PROPERTY IsClosed : BOOL
GET
IF ipTrack <> 0 THEN
	IsClosed := ipTrack.GetIsClosed();
ELSE
	Trace('IsClosed called before initialization!');
	_Error := TRUE;
END_IF
END_GET
END_PROPERTY

PROPERTY Length : LREAL
GET
IF ipTrack <> 0 THEN
	Length := ipTrack.GetLength();
ELSE
	Trace('Length called before initialization!');
	_Error := TRUE;
END_IF
END_GET
END_PROPERTY

PROPERTY Name : STRING
GET
IF ipTrack <> 0 THEN
	Name := ipTrack.GetObjectName();
ELSE
	Trace('Name called before initialization!');
	_Error := TRUE;
END_IF
END_GET
END_PROPERTY

METHOD PRIVATE Initialize : BOOL
CASE InitializeState OF
	E_InitializeState_Track.eInitializeStateTrack_Check:
		IF ipTrack <> 0 THEN
			InitializeState := E_InitializeState_Track.eInitializeStateTrack_GetPartInfo;
		ELSE
			IF Parameters_XTS.ENABLE_DEBUG_TRACING THEN
				Trace('Track initialization attempted with null reference');
			END_IF

			InitializeState := E_InitializeState_Track.eInitializeStateTrack_Failed;
		END_IF

	E_InitializeState_Track.eInitializeStateTrack_GetPartInfo:
		NumberOfParts := ipTrack.GetPartCount();
		Parts		  REF= ipTrack.GetPartInfoItems();
		IF NumberOfParts = 0 THEN
			IF Parameters_XTS.ENABLE_DEBUG_TRACING THEN
				Trace('No parts associated with this track');
			END_IF

			InitializeState := E_InitializeState_Track.eInitializeStateTrack_Failed;
		ELSE
			InitializeState := E_InitializeState_Track.eInitializeStateTrack_Complete;
		END_IF

	E_InitializeState_Track.eInitializeStateTrack_Complete:
		_Busy	   := FALSE;
		Initialize := TRUE;

	E_InitializeState_Track.eInitializeStateTrack_Failed:
		_Busy  := FALSE;
		_Error := TRUE;
END_CASE
END_METHOD

END_FUNCTION_BLOCK

// Utilities/FB_TrackingRegister_Stations
FUNCTION_BLOCK FB_TrackingRegister_Stations
VAR
	Status			 : ARRAY[1..TcIoXtsEnvironmentParameterList.MaxXtsInfoStation] OF BOOL;
	_StationsToTrack : REFERENCE TO UDINT;
END_VAR

//This FB is just for ease of tracking what group commands

//have actually completed

METHOD Check : BOOL
VAR_INPUT
	i : UDINT;
END_VAR
IF __ISVALIDREF(_StationsToTrack) THEN
	IF (i >= 1) AND (i <= _StationsToTrack) THEN
		Check := Status[i];
	END_IF
END_IF
END_METHOD

METHOD Clear : BOOL
MEMSET(ADR(Status), 0, SIZEOF(Status));
END_METHOD

PROPERTY Complete : BOOL
GET
VAR
	i : UDINT;
END_VAR

//Returns true if all operations have completed
IF __ISVALIDREF(_StationsToTrack) THEN
	FOR i := 1 TO _StationsToTrack DO
		IF NOT Status[i] THEN
			Complete := FALSE;
			RETURN;
		END_IF
	END_FOR

	Complete := TRUE;
END_IF
END_GET
END_PROPERTY

PROPERTY NumberCompleted : UDINT
GET
VAR
	i : UDINT;
END_VAR
IF __ISVALIDREF(_StationsToTrack) THEN
	FOR i := 1 TO _StationsToTrack DO
		IF Status[i] THEN
			NumberCompleted := NumberCompleted + 1;
		END_IF
	END_FOR
END_IF
END_GET
END_PROPERTY

METHOD Reset : BOOL
VAR_INPUT
	i : UDINT;
END_VAR
IF __ISVALIDREF(_StationsToTrack) THEN
	IF (i >= 1) AND (i <= _StationsToTrack) THEN
		Status[i] := FALSE;
	END_IF
END_IF
END_METHOD

METHOD Set : BOOL
VAR_INPUT
	i : UDINT;
END_VAR
IF __ISVALIDREF(_StationsToTrack) THEN
	IF (i >= 1) AND (i <= _StationsToTrack) THEN
		Status[i] := TRUE;
	END_IF
END_IF
END_METHOD

PROPERTY StationsToTrack : REFERENCE TO UDINT
GET
StationsToTrack REF= _StationsToTrack;
END_GET
SET
_StationsToTrack REF= StationsToTrack;
END_SET
END_PROPERTY

END_FUNCTION_BLOCK

// XPU/FB_Component_XPU
FUNCTION_BLOCK FINAL FB_Component_XPU EXTENDS FB_ComponentBase IMPLEMENTS I_XTS_Xpu
VAR
	XPUAlarms						: ARRAY[1..CONSTANTS.XPU_ALARM_COUNT] OF FB_TcAlarm;
	CAGroup							: AXES_GROUP_REF; //***Must be linked to the CA group in NC***
	ipXPU							: I_TcIoXtsProcessingUnit;
	ipMc2CAGroup					: I_Mc2CaGroup;
	NumberOfParts					: UDINT;
	Parts							: ARRAY[0..TcIoXtsEnvironmentParameterList.MaxXtsPartsPerXpu] OF FB_XTS_Part;
	NumberOfTracks					: UDINT;
	Tracks							: ARRAY[0..TcIoXtsEnvironmentParameterList.MaxXtsTracksPerXpu] OF FB_XTS_Track;
	NumberOfMovers					: UDINT;
	Movers							: ARRAY[0..TcIoXtsEnvironmentParameterList.MaxXtsMoversPerXpu] OF FB_XTS_Mover;
	ipMovers						: ARRAY[0..TcIoXtsEnvironmentParameterList.MaxXtsMoversPerXpu] OF I_XTS_Mover;
	NumberOfStations				: UDINT;
	InfoStations					: ARRAY[0..TcIoXtsEnvironmentParameterList.MaxXtsInfoServer * TcIoXtsEnvironmentParameterList.MaxXtsInfoStation] OF FB_XTS_InfoStation;
	ipStations						: ARRAY[0..TcIoXtsEnvironmentParameterList.MaxXtsInfoServer * TcIoXtsEnvironmentParameterList.MaxXtsInfoStation] OF I_XTS_ApplicationStation;
	SequenceState					: UDINT;
	InitializeState					: E_XPUInitializeState;
	InitializeState_Environment		: E_XPUInitializeState_Environment;
	InitializeState_XPU				: E_XPUInitializeState_XPU;
	InitializeState_CAGroups		: E_XPUInitializeState_CAGroups;
	InitializeState_InfoStations	: E_XPUInitializeState_InfoStations;
	_State							: E_XTSState;
	MCGroupEnable					: MC_GroupEnable;
	MCGroupDisable					: MC_GroupDisable;
	MCGroupReset					: MC_GroupReset;
	MCGroupStop						: MC_GroupStop;
	MCGroupReadError				: MC_GroupReadError;
	MCGroupReadStatus				: MC_GroupReadStatus;
	MCUngroupAllAxes				: MC_UngroupAllAxes;
	JsonParser						: FB_JsonDomParser;
	MoverTracker					: FB_TrackingRegister_Movers;
	StationTracker					: FB_TrackingRegister_Stations;
	StationRecoveryComplete			: BOOL;
	_MoverAssignmentStorageLocation : E_MoverAssignmentRecoverySource := E_MoverAssignmentRecoverySource.eMoverAssignmentRecoverySource_NoBackup;
	WritePersistentData				: FB_WritePersistentData;
	_PartCoEData					: ARRAY[1..TcIoXtsEnvironmentParameterList.MaxXtsPartsPerXpu] OF ARRAY[1..TcIoXtsEnvironmentParameterList.MaxModulesPerPart] OF ST_AT2xxxAllCoEData;
END_VAR

VAR
	//Upstream/Downstream relationships between stations
	StationNeigbors : ARRAY[0..TcIoXtsEnvironmentParameterList.MaxXtsInfoServer * TcIoXtsEnvironmentParameterList.MaxXtsInfoStation] OF ST_StationNeighbors;
END_VAR

VAR PERSISTENT
	//Power-up mover-station assignments (_MoverAssignmentStorageLocation = E_MoverAssignmentRecoverySource.eMoverAssignmentRecoverySource_Persistent)
	MoverAssignments_Persistent : ARRAY[1..TcIoXtsEnvironmentParameterList.MaxXtsInfoServer * TcIoXtsEnvironmentParameterList.MaxXtsInfoStation] OF ST_MoverAssignmentData;
END_VAR

VAR RETAIN
	//Power-up mover-station assignments (_MoverAssignmentStorageLocation = E_MoverAssignmentRecoverySource.eMoverAssignmentRecoverySource_NOVRAM)
	MoverAssignments_NOVRAM : ARRAY[1..TcIoXtsEnvironmentParameterList.MaxXtsInfoServer * TcIoXtsEnvironmentParameterList.MaxXtsInfoStation] OF ST_MoverAssignmentData;
END_VAR

//! @summary This method serves as the entry point for all underlying FB logic
METHOD PUBLIC CyclicLogic
//! @description This method should be called cyclically by descendant function blocks by invoking <c>SUPER^.CyclicLogic()</c>.  Alternatively, the contents of this method could be reimplemented entirely in which case a call to this method would not be necessary.
VAR
	i, j : UDINT;
END_VAR
SUPER^.CyclicLogic();
IF NOT _InitComplete THEN
	RETURN;
END_IF

FOR i := 1 TO NumberOfParts DO
	Parts[i].CyclicLogic();
	IF NOT InSimulationMode THEN
		_PartCoEData[i] := Parts[i].ModuleCoEData;
	END_IF
END_FOR

FOR i := 1 TO NumberOfTracks DO
	Tracks[i].CyclicLogic();
END_FOR

FOR i := 1 TO NumberOfMovers DO
	IF ipMovers[i] <> 0 THEN
		ipMovers[i].CyclicLogic();
	END_IF

	FOR j := 1 TO NumberOfParts DO
		IF Movers[i].CurrentPartOID = Parts[j].OID THEN
			Movers[i].CurrentPart := Parts[j];
			EXIT;
		END_IF
	END_FOR

	FOR j := 1 TO NumberOfTracks DO
		IF Movers[i].CurrentTrackOID = Tracks[j].OID THEN
			Movers[i].CurrentTrack := Tracks[j];
			EXIT;
		END_IF
	END_FOR
END_FOR

FOR i := 1 TO NumberOfStations DO
	InfoStations[i].CyclicLogic();
END_FOR

IF StationRecoveryComplete THEN
	CollectRecoveryData();
END_IF

(****************    Call misc. group FBs    ****************)
MCGroupEnable(AxesGroup := CAGroup);
MCGroupDisable(AxesGroup := CAGroup);
MCGroupReset(AxesGroup := CAGroup);
MCGroupStop(AxesGroup := CAGroup);
MCUngroupAllAxes(AxesGroup := CAGroup);
MCGroupReadStatus(AxesGroup := CAGroup, Enable := TRUE);
MCGroupReadError(AxesGroup := CAGroup, Enable := TRUE);
_Busy := (_State <> E_XTSState.eXTSState_Disabled) AND (_State <> E_XTSState.eXTSState_Error) AND (_State <> E_XTSState.eXTSState_Enabled);
END_METHOD

METHOD GetPositionOnTrack : LREAL
VAR_INPUT
	TrackID	 : OTCID;
	PartID	 : OTCID;
	Position : LREAL;
END_VAR

VAR
	i			   : UDINT;
	PositionResult : LREAL;
END_VAR
IF TrackID <> 0 THEN
	FOR i := 1 TO NumberOfTracks DO
		IF Tracks[i].OID = TrackID THEN
			Tracks[i].GetTrackPositionByPart(Position, PartID, TrackPosition => GetPositionOnTrack);
			EXIT;
		END_IF
	END_FOR
ELSE
	Tracks[1].GetTrackPositionByPart(Position, PartID, TrackPosition => GetPositionOnTrack);
END_IF
END_METHOD

METHOD GiveMover : BOOL
VAR_INPUT
	RequestingStation : I_XTS_StationNeighbor;
END_VAR

VAR
	i : UDINT;
END_VAR
FOR i := 0 TO NumberOfStations DO
	IF StationNeigbors[i].Station <> 0 THEN
		IF StationNeigbors[i].Station = RequestingStation THEN
			GiveMover := StationNeigbors[i].UpstreamStation.GiveMover(RequestingStation);
			EXIT;
		END_IF
	END_IF
END_FOR
END_METHOD

PROPERTY InSimulationMode : BOOL
GET
IF ipXPU <> 0 THEN
	InSimulationMode := ipXPU.GetOperationMode() = OperationMode.Simulation;
END_IF
END_GET
END_PROPERTY

//! @summary Initializes event function blocks using this components's name
{attribute 'call_after_online_change_slot' := '<slot>'}
METHOD PROTECTED CreateEvents
VAR
	Temp : STRING;
END_VAR
Temp := CONCAT(CONCAT(CONCAT('XPU', ': '), Name),
			   ' '); //Creates a utility string for alarms and other messaging that reads (example text) - "Module 10 - Main Casepacker" to be followed by the alarm or message info

F_CreateAllEventsInClass(Alarms		:= XPUAlarms,
						 ClassSize	:= SIZEOF(TC_EVENTS.XPUAlarms),
						 pInitEvent := ADR(TC_EVENTS.XPUAlarms.InitReferenceEvent),
						 Prefix		:= Name);

SUPER^.CreateEvents();
END_METHOD

//! Provides basic error detection and event handling for this component
METHOD PROTECTED Monitoring
VAR
	i			  : UDINT;
	FaultsCleared : BOOL;
END_VAR
SUPER^.Monitoring();

//ErrorID 2 - Part Error
FaultsCleared := TRUE;
FOR i := 1 TO NumberOfParts DO
	IF Parts[i].Error THEN
		IF NOT XPUAlarms[E_XPUAlarms.PartError].bRaised THEN
			RaiseAlarmWithStrings(XPUAlarms[E_XPUAlarms.PartError], TO_STRING(i), TO_STRING(Parts[i].ErrorID));
			SetError(Parts[i].ErrorID);
			_State := E_XTSState.eXTSState_Error;
		END_IF

		FaultsCleared := FALSE;
		EXIT;
	END_IF
END_FOR

IF XPUAlarms[E_XPUAlarms.PartError].bRaised AND FaultsCleared THEN
	XPUAlarms[E_XPUAlarms.PartError].Clear(0, 0);
END_IF

//ErrorID 3 - Track Error
FaultsCleared := TRUE;
FOR i := 1 TO NumberOfTracks DO
	IF Tracks[i].Error THEN
		IF NOT XPUAlarms[E_XPUAlarms.TrackError].bRaised THEN
			RaiseAlarmWithStrings(XPUAlarms[E_XPUAlarms.TrackError], TO_STRING(i), TO_STRING(Tracks[i].ErrorID));
			SetError(Tracks[i].ErrorID);
			_State := E_XTSState.eXTSState_Error;
		END_IF

		FaultsCleared := FALSE;
		EXIT;
	END_IF
END_FOR

IF XPUAlarms[E_XPUAlarms.TrackError].bRaised AND FaultsCleared THEN
	XPUAlarms[E_XPUAlarms.TrackError].Clear(0, 0);
END_IF

//ErrorID 4 - Mover Error
FaultsCleared := TRUE;
FOR i := 1 TO NumberOfMovers DO
	IF (ipMovers[i] <> 0) AND_THEN ipMovers[i].Error THEN
		IF NOT XPUAlarms[E_XPUAlarms.MoverError].bRaised THEN
			RaiseAlarmWithStrings(XPUAlarms[E_XPUAlarms.MoverError], TO_STRING(i), TO_STRING(ipMovers[i].ErrorID));
			SetError(ipMovers[i].ErrorID);
			_State := E_XTSState.eXTSState_Error;
		END_IF

		FaultsCleared := FALSE;
		EXIT;
	END_IF
END_FOR

IF XPUAlarms[E_XPUAlarms.MoverError].bRaised AND FaultsCleared THEN
	XPUAlarms[E_XPUAlarms.MoverError].Clear(0, 0);
END_IF

//ErrorID 5 - InfoStation Error
FaultsCleared := TRUE;
FOR i := 1 TO NumberOfStations DO
	IF InfoStations[i].Error THEN
		IF NOT XPUAlarms[E_XPUAlarms.InfoStationError].bRaised THEN
			RaiseAlarmWithStrings(XPUAlarms[E_XPUAlarms.InfoStationError], TO_STRING(i), TO_STRING(InfoStations[i].ErrorID));
			SetError(InfoStations[i].ErrorID);
			_State := E_XTSState.eXTSState_Error;
		END_IF

		FaultsCleared := FALSE;
		EXIT;
	END_IF
END_FOR

IF XPUAlarms[E_XPUAlarms.InfoStationError].bRaised AND FaultsCleared THEN
	XPUAlarms[E_XPUAlarms.InfoStationError].Clear(0, 0);
END_IF

//ErrorID 6 - CA Group Error
IF (MCGroupReadError.GroupErrorId <> 0) AND NOT XPUAlarms[E_XPUAlarms.CAGroupError].bRaised THEN
	RaiseAlarmWithStrings(Alarm := XPUAlarms[E_XPUAlarms.CAGroupError], UDINT_TO_STRING(MCGroupReadError.GroupErrorId), '');
	SetError(MCGroupReadError.GroupErrorId);
ELSIF NOT (MCGroupReadError.GroupErrorId <> 0) AND XPUAlarms[E_XPUAlarms.CAGroupError].bRaised THEN
	XPUAlarms[E_XPUAlarms.CAGroupError].Clear(0, 0);
END_IF

//ErrorID 7 - Initialization Error

// This fault is handled in the initialization methods

//ErrorID 8 - MC_GroupEnable Error
IF MCGroupEnable.Error AND NOT XPUAlarms[E_XPUAlarms.GroupEnableError].bRaised THEN
	RaiseAlarmWithStrings(Alarm := XPUAlarms[E_XPUAlarms.GroupEnableError], UDINT_TO_STRING(MCGroupEnable.ErrorID), '');
	SetError(MCGroupEnable.ErrorID);
ELSIF NOT MCGroupEnable.Error AND XPUAlarms[E_XPUAlarms.GroupEnableError].bRaised THEN
	XPUAlarms[E_XPUAlarms.GroupEnableError].Clear(0, 0);
END_IF

//ErrorID 9 - MC_GroupDisable Error
IF MCGroupDisable.Error AND NOT XPUAlarms[E_XPUAlarms.GroupDisableError].bRaised THEN
	RaiseAlarmWithStrings(Alarm := XPUAlarms[E_XPUAlarms.GroupDisableError], UDINT_TO_STRING(MCGroupDisable.ErrorID), '');
	SetError(MCGroupDisable.ErrorID);
ELSIF NOT MCGroupDisable.Error AND XPUAlarms[E_XPUAlarms.GroupDisableError].bRaised THEN
	XPUAlarms[E_XPUAlarms.GroupDisableError].Clear(0, 0);
END_IF

//ErrorID 10 - MC_GroupReset Error
IF MCGroupReset.Error AND NOT XPUAlarms[E_XPUAlarms.GroupResetError].bRaised THEN
	RaiseAlarmWithStrings(Alarm := XPUAlarms[E_XPUAlarms.GroupResetError], UDINT_TO_STRING(MCGroupReset.ErrorID), '');
	SetError(MCGroupReset.ErrorID);
ELSIF NOT MCGroupReset.Error AND XPUAlarms[E_XPUAlarms.GroupResetError].bRaised THEN
	XPUAlarms[E_XPUAlarms.GroupResetError].Clear(0, 0);
END_IF

//ErrorID 11 - MC_GroupStop Error
IF MCGroupStop.Error AND NOT XPUAlarms[E_XPUAlarms.GroupStopError].bRaised THEN
	RaiseAlarmWithStrings(Alarm := XPUAlarms[E_XPUAlarms.GroupStopError], UDINT_TO_STRING(MCGroupStop.ErrorID), '');
	SetError(MCGroupStop.ErrorID);
ELSIF NOT MCGroupStop.Error AND XPUAlarms[E_XPUAlarms.GroupStopError].bRaised THEN
	XPUAlarms[E_XPUAlarms.GroupStopError].Clear(0, 0);
END_IF

//ErrorID 12 - MC_GroupReadError Error
IF MCGroupReadError.Error AND NOT XPUAlarms[E_XPUAlarms.GroupReadErrorError].bRaised THEN
	RaiseAlarmWithStrings(Alarm := XPUAlarms[E_XPUAlarms.GroupReadErrorError], UDINT_TO_STRING(MCGroupReadError.ErrorId), '');
	SetError(MCGroupReadError.ErrorID);
ELSIF NOT MCGroupReadError.Error AND XPUAlarms[E_XPUAlarms.GroupReadErrorError].bRaised THEN
	XPUAlarms[E_XPUAlarms.GroupReadErrorError].Clear(0, 0);
END_IF

//ErrorID 13 - MC_GroupReadStatus Error
IF MCGroupReadStatus.Error AND NOT XPUAlarms[E_XPUAlarms.GroupReadStatusError].bRaised THEN
	RaiseAlarmWithStrings(Alarm := XPUAlarms[E_XPUAlarms.GroupReadStatusError], UDINT_TO_STRING(MCGroupReadStatus.ErrorID), '');
	SetError(MCGroupReadStatus.ErrorID);
ELSIF NOT MCGroupReadStatus.Error AND XPUAlarms[E_XPUAlarms.GroupReadStatusError].bRaised THEN
	XPUAlarms[E_XPUAlarms.GroupReadStatusError].Clear(0, 0);
END_IF

//ErrorID 14 - MC_UngroupAllAxes Error
IF MCUngroupAllAxes.Error AND NOT XPUAlarms[E_XPUAlarms.UngroupAllAxesError].bRaised THEN
	RaiseAlarmWithStrings(Alarm := XPUAlarms[E_XPUAlarms.UngroupAllAxesError], UDINT_TO_STRING(MCUngroupAllAxes.ErrorID), '');
	SetError(MCUngroupAllAxes.ErrorID);
ELSIF NOT MCUngroupAllAxes.Error AND XPUAlarms[E_XPUAlarms.UngroupAllAxesError].bRaised THEN
	XPUAlarms[E_XPUAlarms.UngroupAllAxesError].Clear(0, 0);
END_IF

_CurrentAlarmSeverity := F_GetMaxSeverityRaised(Alarms := XPUAlarms, CurrentSeverity := CurrentAlarmSeverity);
END_METHOD

METHOD PRIVATE Initialize_CAGroups : BOOL
VAR
	i : UDINT;
END_VAR
CASE InitializeState_CAGroups OF
	E_XPUInitializeState_CAGroups.eXPUInitializeStateCAGroups_CheckMapping:
		//Ensure the CA group variable is linked to the TcCom object
		IF F_GetMappingStatus(ADR(CAGroup.NcToPlc), SIZEOF(CAGroup.NcToPlc)) <> EPlcMappingStatus.MS_Mapped THEN
			IF Parameters_XTS.ENABLE_DEBUG_TRACING THEN
				Trace('CA Group NcToPlc not mapped');
			END_IF

			InitializeState_CAGroups := E_XPUInitializeState_CAGroups.eXPUInitializeStateCAGroups_Failed;
		ELSIF F_GetMappingStatus(ADR(CAGroup.PlcToNc), SIZEOF(CAGroup.PlcToNc)) <> EPlcMappingStatus.MS_Mapped THEN
			IF Parameters_XTS.ENABLE_DEBUG_TRACING THEN
				Trace('CA Group PlcToNc not mapped');
			END_IF

			InitializeState_CAGroups := E_XPUInitializeState_CAGroups.eXPUInitializeStateCAGroups_Failed;
		ELSE
			InitializeState_CAGroups := E_XPUInitializeState_CAGroups.eXPUInitializeStateCAGroups_FindGroupID;
		END_IF

	E_XPUInitializeState_CAGroups.eXPUInitializeStateCAGroups_FindGroupID:
		//Find the correct CA group OID for this XTS and assign the interface
		FOR i := 1 TO TcIoXtsEnvironmentParameterList.MaxXtsCaGroup DO
			IF CAGroup.NcToPlc.Common.GroupOID = XTS.CAGroupOIDs[i] THEN
				ipMc2CAGroup := XTS.Environment.Mc2CaGroup(TO_UINT(i));
				EXIT;
			END_IF
		END_FOR

		IF ipMc2CAGroup <> 0 THEN
			InitializeState_CAGroups := E_XPUInitializeState_CAGroups.eXPUInitializeStateCAGroups_CheckGroupInitialized;
		ELSE
			IF Parameters_XTS.ENABLE_DEBUG_TRACING THEN
				Trace('No matching CA group found in XTS environment');
			END_IF

			InitializeState_CAGroups := E_XPUInitializeState_CAGroups.eXPUInitializeStateCAGroups_Failed;
		END_IF

	E_XPUInitializeState_CAGroups.eXPUInitializeStateCAGroups_CheckGroupInitialized:
		IF ipMc2CAGroup.P_IsInitialized THEN
			IF Parameters_XTS.ENABLE_DEBUG_TRACING THEN
				Trace('CA Group Initialized');
			END_IF

			InitializeState_CAGroups := E_XPUInitializeState_CAGroups.eXPUInitializeStateCAGroups_Complete;
		ELSE
			IF Parameters_XTS.ENABLE_DEBUG_TRACING THEN
				Trace('CA group environment FB not initialized');
			END_IF

			InitializeState_CAGroups := E_XPUInitializeState_CAGroups.eXPUInitializeStateCAGroups_Failed;
		END_IF

	E_XPUInitializeState_CAGroups.eXPUInitializeStateCAGroups_Complete:
		Initialize_CAGroups := TRUE;

	E_XPUInitializeState_CAGroups.eXPUInitializeStateCAGroups_Failed:
		IF NOT XPUAlarms[E_XPUAlarms.InitializationError].bRaised THEN
			RaiseAlarm(Alarm := XPUAlarms[E_XPUAlarms.InitializationError]);
		END_IF
END_CASE
END_METHOD

METHOD PRIVATE Initialize_Environment : BOOL
CASE InitializeState_Environment OF
	E_XPUInitializeState_Environment.eXPUInitializeStateEnvironment_Check:
		IF XTS.InitializationComplete THEN
			IF Parameters_XTS.ENABLE_DEBUG_TRACING THEN
				Trace('XTS environment already initialized');
			END_IF

			InitializeState_Environment := E_XPUInitializeState_Environment.eXPUInitializeStateEnvironment_Complete;
		ELSE
			IF XTS.InitializationInProgress THEN
				IF Parameters_XTS.ENABLE_DEBUG_TRACING THEN
					Trace('XTS environment initialization in progress already');
				END_IF

				InitializeState_Environment := E_XPUInitializeState_Environment.eXPUInitializeStateEnvironment_WaitingForOtherXTS;
			ELSE
				IF Parameters_XTS.ENABLE_DEBUG_TRACING THEN
					Trace('Initializing XTS environment');
				END_IF

				XTS.Environment.P_XtsEnvironmentConfiguration := XTS.XTSEnvironmentConfig;
				XTS.InitializationInProgress				  := TRUE;
				InitializeState_Environment					  := E_XPUInitializeState_Environment.eXPUInitializeStateEnvironment_InitializeEnvironment;
			END_IF
		END_IF

	E_XPUInitializeState_Environment.eXPUInitializeStateEnvironment_InitializeEnvironment:
		IF XTS.Environment.Init(TRUE) THEN
			XTS.Environment.Init(FALSE);
			IF XTS.Environment.P_IsInitialized THEN
				InitializeState_Environment := E_XPUInitializeState_Environment.eXPUInitializeStateEnvironment_GetXPUCount;
			ELSE
				IF Parameters_XTS.ENABLE_DEBUG_TRACING THEN
					Trace('XTS environment initialization failed');
				END_IF

				InitializeState_Environment := E_XPUInitializeState_Environment.eXPUInitializeStateEnvironment_Failed;
			END_IF
		ELSIF XTS.Environment.bError THEN
			IF Parameters_XTS.ENABLE_DEBUG_TRACING THEN
				Trace('XTS environment initialization failed');
			END_IF

			InitializeState_Environment := E_XPUInitializeState_Environment.eXPUInitializeStateEnvironment_Failed;
		END_IF

	E_XPUInitializeState_Environment.eXPUInitializeStateEnvironment_GetXPUCount:
		IF XTS.XTSEnvironmentConfig.bEnableInitXpu THEN
			IF XTS.Environment.GetXpuCount(TRUE) THEN
				XTS.Environment.GetXpuCount(FALSE);
				XTS.XPUCount := XTS.Environment.P_XpuCountUint;
				IF Parameters_XTS.ENABLE_DEBUG_TRACING THEN
					Trace(CONCAT('Found ', CONCAT(TO_STRING(XTS.XPUCount), ' XPUs')));
				END_IF

				InitializeState_Environment := E_XPUInitializeState_Environment.eXPUInitializeStateEnvironment_GetXPUOIDs;
			END_IF
		ELSE
			IF Parameters_XTS.ENABLE_DEBUG_TRACING THEN
				Trace('XPUs disabled in environment configuration');
			END_IF

			InitializeState_Environment := E_XPUInitializeState_Environment.eXPUInitializeStateEnvironment_GetInfoServerCounts;
		END_IF

	E_XPUInitializeState_Environment.eXPUInitializeStateEnvironment_GetXPUOIDs:
		IF XTS.XPUCount > 0 THEN
			IF XTS.Environment.GetXpuOids(TRUE) THEN
				XTS.Environment.GetXpuOids(FALSE);
				XTS.XPUOIDs					REF= XTS.Environment.P_XpuOids;
				InitializeState_Environment := E_XPUInitializeState_Environment.eXPUInitializeStateEnvironment_GetInfoServerCounts;
			END_IF
		ELSE
			IF Parameters_XTS.ENABLE_DEBUG_TRACING THEN
				Trace('No XPUs found');
			END_IF

			InitializeState_Environment := E_XPUInitializeState_Environment.eXPUInitializeStateEnvironment_GetInfoServerCounts;
		END_IF

	E_XPUInitializeState_Environment.eXPUInitializeStateEnvironment_GetInfoServerCounts:
		IF XTS.XTSEnvironmentConfig.bEnableInitInfoServer THEN
			IF XTS.Environment.GetInfoServerCount(TRUE) THEN
				XTS.Environment.GetInfoServerCount(FALSE);
				XTS.InfoServerCount := XTS.Environment.P_InfoServerCount;
				IF Parameters_XTS.ENABLE_DEBUG_TRACING THEN
					Trace(CONCAT('Found ', CONCAT(TO_STRING(XTS.InfoServerCount), ' InfoServer(s)')));
				END_IF

				InitializeState_Environment := E_XPUInitializeState_Environment.eXPUInitializeStateEnvironment_GetInfoServerOIDs;
			END_IF
		ELSE
			IF Parameters_XTS.ENABLE_DEBUG_TRACING THEN
				Trace('InfoServers disabled in environment configuration');
			END_IF

			InitializeState_Environment := E_XPUInitializeState_Environment.eXPUInitializeStateEnvironment_GetCAGroupCounts;
		END_IF

	E_XPUInitializeState_Environment.eXPUInitializeStateEnvironment_GetInfoServerOIDs:
		IF XTS.InfoServerCount > 0 THEN
			XTS.InfoServerOIDs			REF= XTS.Environment.P_InfoServerOids;
			InitializeState_Environment := E_XPUInitializeState_Environment.eXPUInitializeStateEnvironment_GetCAGroupCounts;
		ELSE
			IF Parameters_XTS.ENABLE_DEBUG_TRACING THEN
				Trace('No InfoServers found');
			END_IF

			InitializeState_Environment := E_XPUInitializeState_Environment.eXPUInitializeStateEnvironment_GetCAGroupCounts;
		END_IF

	E_XPUInitializeState_Environment.eXPUInitializeStateEnvironment_GetCAGroupCounts:
		IF XTS.XTSEnvironmentConfig.bEnableInitCaGroup THEN
			IF XTS.Environment.GetCaGroupCount(TRUE) THEN
				XTS.Environment.GetCaGroupCount(FALSE);
				XTS.CAGroupCount := XTS.Environment.P_CaGroupCount;
				IF Parameters_XTS.ENABLE_DEBUG_TRACING THEN
					Trace(CONCAT('Found ', CONCAT(TO_STRING(XTS.CAGroupCount), ' CA group(s)')));
				END_IF

				InitializeState_Environment := E_XPUInitializeState_Environment.eXPUInitializeStateEnvironment_GetCAGroupOIDs;
			END_IF
		ELSE
			IF Parameters_XTS.ENABLE_DEBUG_TRACING THEN
				Trace('CA Groups disabled in environment configuration');
			END_IF

			InitializeState_Environment := E_XPUInitializeState_Environment.eXPUInitializeStateEnvironment_Cleanup;
		END_IF

	E_XPUInitializeState_Environment.eXPUInitializeStateEnvironment_GetCAGroupOIDs:
		IF XTS.CAGroupCount > 0 THEN
			IF XTS.Environment.GetCaGroupOids(TRUE) THEN
				XTS.Environment.GetCaGroupOids(FALSE);
				XTS.CAGroupOIDs				REF= XTS.Environment.P_CaGroupOids;
				InitializeState_Environment := E_XPUInitializeState_Environment.eXPUInitializeStateEnvironment_Cleanup;
			END_IF
		ELSE
			IF Parameters_XTS.ENABLE_DEBUG_TRACING THEN
				Trace('No CA groups found');
			END_IF

			InitializeState_Environment := E_XPUInitializeState_Environment.eXPUInitializeStateEnvironment_Cleanup;
		END_IF

	E_XPUInitializeState_Environment.eXPUInitializeStateEnvironment_Cleanup:
		IF Parameters_XTS.ENABLE_DEBUG_TRACING THEN
			Trace('XTS environment initialization complete');
		END_IF

		XTS.InitializationInProgress := FALSE;
		XTS.InitializationComplete	 := TRUE;
		InitializeState_Environment	 := E_XPUInitializeState_Environment.eXPUInitializeStateEnvironment_Complete;

	E_XPUInitializeState_Environment.eXPUInitializeStateEnvironment_WaitingForOtherXTS:
		//Holding state in case of multiple XTS and init already in progress
		IF XTS.InitializationComplete THEN
			InitializeState_Environment := E_XPUInitializeState_Environment.eXPUInitializeStateEnvironment_Complete;
		END_IF

	E_XPUInitializeState_Environment.eXPUInitializeStateEnvironment_Complete:
		Initialize_Environment := TRUE;

	E_XPUInitializeState_Environment.eXPUInitializeStateEnvironment_Failed:
		IF NOT XPUAlarms[E_XPUAlarms.InitializationError].bRaised THEN
			RaiseAlarm(Alarm := XPUAlarms[E_XPUAlarms.InitializationError]);
		END_IF
END_CASE
END_METHOD

METHOD Initialize_InfoStations : BOOL
VAR
	i, j, k, l		 : UDINT;
	StationPartCount : UDINT;
	StationPartOIDs	 : REFERENCE TO ARRAY[1..TcIoXtsEnvironmentParameterList.MaxXtsPartsPerXpu] OF OTCID;
	StationMatched	 : BOOL;
END_VAR

VAR_INST
	OIDs_Parts : REFERENCE TO ARRAY[1..TcIoXtsEnvironmentParameterList.MaxXtsPartsPerXpu] OF OTCID;
END_VAR
CASE InitializeState_InfoStations OF
	E_XPUInitializeState_InfoStations.eXPUInitializeStateInfoStations_GetInfoServerInterfaces:
		//Collect interface pointers for all InfoServers
		FOR i := 1 TO XTS.InfoServerCount DO
			XTS.ipInfoServer[i] := XTS.Environment.InfoServerTcIo(TO_UINT(i));
			IF XTS.ipInfoServer[i] <> 0 THEN
				IF NOT XTS.ipInfoServer[i].P_IsInitialized THEN
					IF Parameters_XTS.ENABLE_DEBUG_TRACING THEN
						Trace(CONCAT('InfoServer ', CONCAT(TO_STRING(i), ' is not initialized.')));
					END_IF

					InitializeState_InfoStations := E_XPUInitializeState_InfoStations.eXPUInitializeStateInfoStations_Failed;
					RETURN;
				END_IF
			ELSE
				IF Parameters_XTS.ENABLE_DEBUG_TRACING THEN
					Trace(CONCAT('InfoServer ', CONCAT(TO_STRING(i), ' did not return a valid interface')));
				END_IF

				InitializeState_InfoStations := E_XPUInitializeState_InfoStations.eXPUInitializeStateInfoStations_Failed;
				RETURN;
			END_IF
		END_FOR

		InitializeState_InfoStations := E_XPUInitializeState_InfoStations.eXPUInitializeStateInfoStations_GetPartOIDs;

	E_XPUInitializeState_InfoStations.eXPUInitializeStateInfoStations_GetPartOIDs:
		//Collect OIDs for all parts in this XPU--we will use these to match against InfoStations
		OIDs_Parts REF= ipXPU.P_PartOids;
		IF NOT __ISVALIDREF(OIDs_Parts) THEN
			IF Parameters_XTS.ENABLE_DEBUG_TRACING THEN
				Trace('XPU returned an invalid reference');
			END_IF

			InitializeState_XPU := E_XPUInitializeState_XPU.eXPUInitializeStateXPU_Failed;
			RETURN;
		END_IF

		InitializeState_InfoStations := E_XPUInitializeState_InfoStations.eXPUInitializeStateInfoStations_GetStationCounts;

	E_XPUInitializeState_InfoStations.eXPUInitializeStateInfoStations_GetStationCounts:
		//Get the number of InfoStations assocciated with each InfoServer
		FOR i := 1 TO XTS.InfoServerCount DO
			XTS.InfoStationCounts[i] := XTS.ipInfoServer[i].GetInfoStationCount();
		END_FOR

		InitializeState_InfoStations := E_XPUInitializeState_InfoStations.eXPUInitializeStateInfoStations_GetStationInterfaces;

	E_XPUInitializeState_InfoStations.eXPUInitializeStateInfoStations_GetStationInterfaces:
		//Iterate through all InfoServers and InfoStations
		FOR i := 1 TO XTS.InfoServerCount DO
			FOR j := 1 TO XTS.InfoStationCounts[i] DO
				//Store interface pointer to this InfoStation
				XTS.ipInfoStations[i, j] := XTS.ipInfoServer[i].InfoStationTcIo(TO_UINT(j));
				IF XTS.ipInfoStations[i, j] <> 0 THEN
					IF NOT XTS.ipInfoStations[i, j].P_IsInitialized THEN
						IF Parameters_XTS.ENABLE_DEBUG_TRACING THEN
							Trace(CONCAT('InfoStation ', CONCAT(TO_STRING(i), CONCAT(', InfoStation ', CONCAT(TO_STRING(j), ' is not initialized')))));
						END_IF

						InitializeState_InfoStations := E_XPUInitializeState_InfoStations.eXPUInitializeStateInfoStations_Failed;
						RETURN;
					END_IF
				ELSE
					IF Parameters_XTS.ENABLE_DEBUG_TRACING THEN
						Trace(CONCAT('InfoStation ', CONCAT(TO_STRING(i), CONCAT(', InfoStation ', CONCAT(TO_STRING(j), ' did not return a valid interface')))));
					END_IF

					InitializeState_InfoStations := E_XPUInitializeState_InfoStations.eXPUInitializeStateInfoStations_Failed;
					RETURN;
				END_IF
			END_FOR
		END_FOR

		InitializeState_InfoStations := E_XPUInitializeState_InfoStations.eXPUInitializeStateInfoStations_MatchStationsAgainstParts;

	E_XPUInitializeState_InfoStations.eXPUInitializeStateInfoStations_MatchStationsAgainstParts:
		//XPU initialization must be enabled in environment to get part info to match against
		IF XTS.XTSEnvironmentConfig.bEnableInitXpu THEN
			//Loop through all InfoServers
			FOR i := 1 TO XTS.InfoServerCount DO
				//Loop through all InfoStations associated with this InfoServer
				FOR j := 1 TO XTS.InfoStationCounts[i] DO
					StationMatched := FALSE;

					//Get number of parts associated with this station
					StationPartCount := XTS.ipInfoStations[i, j].GetPartCount();
					IF StationPartCount > 0 THEN
						//Get the OIDs of all the parts associated with this station
						StationPartOIDs REF= XTS.ipInfoStations[i, j].GetPartObjectIds();
						IF __ISVALIDREF(StationPartOIDs) THEN
							//Loop through all of the parts associated with this XPU
							FOR k := 1 TO ipXPU.GetPartCount() DO
								FOR l := 1 TO StationPartCount DO
									IF StationPartOIDs[l] = OIDs_Parts[k] THEN
										StationMatched := TRUE;
										EXIT;
									END_IF
								END_FOR

								IF StationMatched THEN
									NumberOfStations							 := NumberOfStations + 1;
									InfoStations[NumberOfStations].ipInfoStation := XTS.ipInfoStations[i, j];
									InfoStations[NumberOfStations].ipXPU		 := THIS^;
									IF NOT (ipStations[NumberOfStations] <> 0) THEN
										IF Parameters_XTS.ENABLE_DEBUG_TRACING THEN
											Trace(CONCAT('No equipment module assigned to slot ', TO_STRING(NumberOfStations)));
										END_IF

										InitializeState_InfoStations := E_XPUInitializeState_InfoStations.eXPUInitializeStateInfoStations_Failed;
										RETURN;
									ELSE
										ipStations[NumberOfStations].InfoStation := InfoStations[NumberOfStations];
										SetStationNeighbors();
										EXIT;
									END_IF
								END_IF
							END_FOR
						ELSE
							IF Parameters_XTS.ENABLE_DEBUG_TRACING THEN
								Trace(CONCAT('InfoStation ', CONCAT(TO_STRING(i), CONCAT(', InfoStation ', CONCAT(TO_STRING(j), ' returned an invalid reference')))));
							END_IF

							InitializeState_InfoStations := E_XPUInitializeState_InfoStations.eXPUInitializeStateInfoStations_Failed;
							RETURN;
						END_IF
					END_IF
				END_FOR
			END_FOR
		ELSE
			IF Parameters_XTS.ENABLE_DEBUG_TRACING THEN
				Trace('XPU initialization was disabled.  Part info needed to match InfoStations.');
			END_IF
		END_IF

		InitializeState_InfoStations := E_XPUInitializeState_InfoStations.eXPUInitializeStateInfoStations_Complete;

	E_XPUInitializeState_InfoStations.eXPUInitializeStateInfoStations_Complete:
		Initialize_InfoStations := TRUE;

	E_XPUInitializeState_InfoStations.eXPUInitializeStateInfoStations_Failed:
		IF NOT XPUAlarms[E_XPUAlarms.InitializationError].bRaised THEN
			RaiseAlarm(Alarm := XPUAlarms[E_XPUAlarms.InitializationError]);
		END_IF
END_CASE
END_METHOD

METHOD Initialize_XPU : BOOL
VAR_INST
	XPUId : UINT;
END_VAR

VAR
	FoundLinkedAxis : BOOL;
	i				: UDINT;
	ipPart			: I_TcIoXtsXpuPart;
	ipMover			: I_TcIoXtsXpuMover;
	ipTrack			: I_TcIoXtsXpuTrack;
END_VAR
CASE InitializeState_XPU OF
	E_XPUInitializeState_XPU.eXPUInitializeStateXPU_FindLinkedMover:
		//Find first available mover FB that is linked to the NC
		FOR i := 1 TO TcIoXtsEnvironmentParameterList.MaxXtsMoversPerXpu DO
			IF Movers[i].AxisRefLinked THEN
				FoundLinkedAxis := TRUE;
				EXIT;
			END_IF
		END_FOR

		IF FoundLinkedAxis THEN
			IF Parameters_XTS.ENABLE_DEBUG_TRACING THEN
				Trace(CONCAT('Using axis ID ', CONCAT(TO_STRING(i), ' to determind XPU ID')));
			END_IF

			InitializeState_XPU := E_XPUInitializeState_XPU.eXPUInitializeStateXPU_FindXPUId;
		ELSE
			IF Parameters_XTS.ENABLE_DEBUG_TRACING THEN
				Trace('No linked axes found!');
			END_IF

			InitializeState_XPU := E_XPUInitializeState_XPU.eXPUInitializeStateXPU_Failed;
		END_IF

	E_XPUInitializeState_XPU.eXPUInitializeStateXPU_FindXPUId:
		//Get the correct XPU ID via the first linked mover
		XPUId := XTS.Environment.GetXpuNumberByAxisId(Movers[1].Axis.NcToPlc.AxisId);
		IF XPUId <> 0 THEN
			IF XPUId < 1 OR XPUId > XTS.XPUCount THEN
				IF Parameters_XTS.ENABLE_DEBUG_TRACING THEN
					Trace('Invalid XPU ID found');
				END_IF

				InitializeState_XPU := E_XPUInitializeState_XPU.eXPUInitializeStateXPU_Failed;
			ELSE
				IF Parameters_XTS.ENABLE_DEBUG_TRACING THEN
					Trace(CONCAT('Found XPU ID ', (TO_STRING(i))));
				END_IF

				InitializeState_XPU := E_XPUInitializeState_XPU.eXPUInitializeStateXPU_GetXPUInterface;
			END_IF
		ELSE
			IF Parameters_XTS.ENABLE_DEBUG_TRACING THEN
				Trace('No corresponding XPU found');
			END_IF

			InitializeState_XPU := E_XPUInitializeState_XPU.eXPUInitializeStateXPU_Failed;
		END_IF

	E_XPUInitializeState_XPU.eXPUInitializeStateXPU_GetXPUInterface:
		//Get interface pointer for the XPU that corresponds to the above XPU ID
		ipXPU := XTS.Environment.XpuTcIo(XPUId);
		IF ipXPU <> 0 THEN
			InitializeState_XPU := E_XPUInitializeState_XPU.eXPUInitializeStateXPU_GetPartCount;
		ELSE
			IF Parameters_XTS.ENABLE_DEBUG_TRACING THEN
				Trace(CONCAT('XPU number ', CONCAT(TO_STRING(XPUId), ' did not return a valid interface')));
			END_IF

			InitializeState_XPU := E_XPUInitializeState_XPU.eXPUInitializeStateXPU_Failed;
		END_IF

	E_XPUInitializeState_XPU.eXPUInitializeStateXPU_GetPartCount:
		//Store the number of PARTS that is associated with this XPU
		NumberOfParts := ipXPU.GetPartCount();
		IF NumberOfParts > 0 THEN
			InitializeState_XPU := E_XPUInitializeState_XPU.eXPUInitializeStateXPU_GetPartInterfaces;
		ELSE
			IF Parameters_XTS.ENABLE_DEBUG_TRACING THEN
				Trace('XPU reports no parts available');
			END_IF

			InitializeState_XPU := E_XPUInitializeState_XPU.eXPUInitializeStateXPU_GetTrackCount;
		END_IF

	E_XPUInitializeState_XPU.eXPUInitializeStateXPU_GetPartInterfaces:
		//Get interface pointers for all PARTS associated with this XPU
		FOR i := 1 TO NumberOfParts DO
			ipPart := ipXPU.PartTcIo(TO_UINT(i));
			IF ipPart <> 0 THEN
				IF NOT ipPart.P_IsInitialized THEN
					IF Parameters_XTS.ENABLE_DEBUG_TRACING THEN
						Trace(CONCAT('Part number ', CONCAT(TO_STRING(i), ' is not initialized.')));
					END_IF

					InitializeState_XPU := E_XPUInitializeState_XPU.eXPUInitializeStateXPU_Failed;
					RETURN;
				ELSE
					Parts[i].ipPart := ipPart;
					Parts[i].OID	:= ipXPU.P_PartOids[i];
				END_IF
			ELSE
				IF Parameters_XTS.ENABLE_DEBUG_TRACING THEN
					Trace(CONCAT('Part number ', CONCAT(TO_STRING(i), ' did not return a valid interface')));
				END_IF

				InitializeState_XPU := E_XPUInitializeState_XPU.eXPUInitializeStateXPU_Failed;
				RETURN;
			END_IF
		END_FOR

		InitializeState_XPU := E_XPUInitializeState_XPU.eXPUInitializeStateXPU_GetTrackCount;

	E_XPUInitializeState_XPU.eXPUInitializeStateXPU_GetTrackCount:
		//Store the number of TRACKS that is associated with this XPU
		NumberOfTracks := ipXPU.GetTrackCount();
		IF NumberOfTracks > 0 THEN
			InitializeState_XPU := E_XPUInitializeState_XPU.eXPUInitializeStateXPU_GetTrackInterfaces;
		ELSE
			IF Parameters_XTS.ENABLE_DEBUG_TRACING THEN
				Trace('XPU reports no tracks available');
			END_IF

			InitializeState_XPU := E_XPUInitializeState_XPU.eXPUInitializeStateXPU_Failed;
		END_IF

	E_XPUInitializeState_XPU.eXPUInitializeStateXPU_GetTrackInterfaces:
		//Get interface pointers for all TRACKS associated with this XPU
		FOR i := 1 TO NumberOfTracks DO
			ipTrack := ipXPU.TrackTcIo(TO_UINT(i));
			IF ipTrack <> 0 THEN
				IF NOT ipTrack.P_IsInitialized THEN
					IF Parameters_XTS.ENABLE_DEBUG_TRACING THEN
						Trace(CONCAT('Track number ', CONCAT(TO_STRING(i), ' is not initialized.')));
					END_IF

					InitializeState_XPU := E_XPUInitializeState_XPU.eXPUInitializeStateXPU_Failed;
					RETURN;
				ELSE
					Tracks[i].ipTrack := ipTrack;
					Tracks[i].OID	  := ipXPU.P_TrackOids[i];
				END_IF
			ELSE
				IF Parameters_XTS.ENABLE_DEBUG_TRACING THEN
					Trace(CONCAT('Track number ', CONCAT(TO_STRING(i), ' did not return a valid interface')));
				END_IF

				InitializeState_XPU := E_XPUInitializeState_XPU.eXPUInitializeStateXPU_Failed;
				RETURN;
			END_IF
		END_FOR

		InitializeState_XPU := E_XPUInitializeState_XPU.eXPUInitializeStateXPU_GetMoverCount;

	E_XPUInitializeState_XPU.eXPUInitializeStateXPU_GetMoverCount:
		//Store the number of MOVERS that is associated with this XPU
		NumberOfMovers := ipXPU.GetMoverCount();
		IF NumberOfMovers > 0 THEN
			InitializeState_XPU := E_XPUInitializeState_XPU.eXPUInitializeStateXPU_GetMoverInterfaces;
		ELSE
			IF Parameters_XTS.ENABLE_DEBUG_TRACING THEN
				Trace('XPU reports no movers available');
			END_IF

			InitializeState_XPU := E_XPUInitializeState_XPU.eXPUInitializeStateXPU_Complete;
		END_IF

	E_XPUInitializeState_XPU.eXPUInitializeStateXPU_GetMoverInterfaces:
		//Get interface pointers for all MOVERS associated with this XPU
		FOR i := 1 TO NumberOfMovers DO
			ipMover := ipXPU.MoverTcIo(TO_UINT(i));
			IF ipMover <> 0 THEN
				IF NOT ipMover.P_IsInitialized THEN
					IF Parameters_XTS.ENABLE_DEBUG_TRACING THEN
						Trace(CONCAT('Mover number ', CONCAT(TO_STRING(i), ' is not initialized.')));
					END_IF

					InitializeState_XPU := E_XPUInitializeState_XPU.eXPUInitializeStateXPU_Failed;
					RETURN;
				ELSE
					Movers[i].ipMover := ipMover;
				END_IF
			ELSE
				IF Parameters_XTS.ENABLE_DEBUG_TRACING THEN
					Trace(CONCAT('Mover number ', CONCAT(TO_STRING(i), ' did not return a valid interface')));
				END_IF

				InitializeState_XPU := E_XPUInitializeState_XPU.eXPUInitializeStateXPU_Failed;
				RETURN;
			END_IF
		END_FOR

		InitializeState_XPU := E_XPUInitializeState_XPU.eXPUInitializeStateXPU_Complete;

	E_XPUInitializeState_XPU.eXPUInitializeStateXPU_Complete:
		//Initialization state complete
		Initialize_XPU := TRUE;

	E_XPUInitializeState_XPU.eXPUInitializeStateXPU_Failed:
		IF NOT XPUAlarms[E_XPUAlarms.InitializationError].bRaised THEN
			RaiseAlarm(Alarm := XPUAlarms[E_XPUAlarms.InitializationError]);
		END_IF
END_CASE
END_METHOD

//! @summary Basic component initialization logic
METHOD PROTECTED Initialize : BOOL;
VAR
	i				  : UDINT;
	AllFBsInitialized : BOOL;
END_VAR

//! @description This method is called by <c>CyclicLogic()</c> as required
CASE InitializeState OF
	E_XPUInitializeState.eXPUInitializeState_Environment:
		IF Initialize_Environment() THEN
			InitializeState := E_XPUInitializeState.eXPUInitializeState_CAGroups;
		END_IF

	E_XPUInitializeState.eXPUInitializeState_CAGroups:
		IF XTS.XTSEnvironmentConfig.bEnableInitCaGroup THEN
			IF Initialize_CAGroups() THEN
				InitializeState := E_XPUInitializeState.eXPUInitializeState_XPU;
			END_IF
		ELSE
			InitializeState := E_XPUInitializeState.eXPUInitializeState_XPU;
		END_IF

	E_XPUInitializeState.eXPUInitializeState_XPU:
		IF XTS.XTSEnvironmentConfig.bEnableInitXpu THEN
			IF Initialize_XPU() THEN
				InitializeState := E_XPUInitializeState.eXPUInitializeState_InfoStations;
			END_IF
		ELSE
			InitializeState := E_XPUInitializeState.eXPUInitializeState_InfoStations;
		END_IF

	E_XPUInitializeState.eXPUInitializeState_InfoStations:
		IF XTS.XTSEnvironmentConfig.bEnableInitInfoServer THEN
			IF Initialize_InfoStations() THEN
				InitializeState := E_XPUInitializeState.eXPUInitializeState_Parts;
			END_IF
		ELSE
			InitializeState := E_XPUInitializeState.eXPUInitializeState_Parts;
		END_IF

	E_XPUInitializeState.eXPUInitializeState_Parts:
		IF XTS.XTSEnvironmentConfig.bEnableInitXpu THEN
			AllFBsInitialized := TRUE;
			FOR i := 1 TO NumberOfParts DO
				IF NOT Parts[i].InitComplete THEN
					AllFBsInitialized := FALSE;
					Parts[i].CyclicLogic();
				END_IF
			END_FOR

			IF AllFBsInitialized THEN
				InitializeState := E_XPUInitializeState.eXPUInitializeState_Tracks;
			END_IF
		ELSE
			//There will be no part information unless the XPU was initialized
			InitializeState := E_XPUInitializeState.eXPUInitializeState_Complete;
		END_IF

	E_XPUInitializeState.eXPUInitializeState_Tracks:
		IF XTS.XTSEnvironmentConfig.bEnableInitXpu THEN
			AllFBsInitialized := TRUE;
			FOR i := 1 TO NumberOfTracks DO
				IF NOT Tracks[i].InitComplete THEN
					AllFBsInitialized := FALSE;
					Tracks[i].CyclicLogic();
				END_IF
			END_FOR

			IF AllFBsInitialized THEN
				FOR i := 1 TO NumberOfTracks DO
					IF (ipMc2CAGroup <> 0) AND_THEN (ipMc2CAGroup.GetRailLength() <> Tracks[i].Length) THEN
						Trace(CONCAT('Track ', CONCAT(TO_STRING(i), ' length does not match CA group rail length!!')));
					END_IF
				END_FOR

				InitializeState := E_XPUInitializeState.eXPUInitializeState_Movers;
			END_IF
		ELSE
			//There will be no track information unless the XPU was initialized
			InitializeState := E_XPUInitializeState.eXPUInitializeState_Complete;
		END_IF

	E_XPUInitializeState.eXPUInitializeState_Movers:
		IF XTS.XTSEnvironmentConfig.bEnableInitXpu THEN
			AllFBsInitialized := TRUE;
			FOR i := 1 TO NumberOfMovers DO
				IF Movers[i].Error THEN
					InitializeState := E_XPUInitializeState.eXPUInitializeState_Failed;
					RETURN;
				ELSIF NOT Movers[i].InitComplete THEN
					AllFBsInitialized := FALSE;
					Movers[i].CyclicLogic();
				END_IF
			END_FOR

			IF AllFBsInitialized THEN
				InitializeState := E_XPUInitializeState.eXPUInitializeState_Stations;
			END_IF
		ELSE
			//There will be no mover information unless the XPU was initialized
			InitializeState := E_XPUInitializeState.eXPUInitializeState_Complete;
		END_IF

	E_XPUInitializeState.eXPUInitializeState_Stations:
		IF XTS.XTSEnvironmentConfig.bEnableInitXpu THEN
			AllFBsInitialized := TRUE;
			FOR i := 1 TO NumberOfStations DO
				IF NOT InfoStations[i].InitComplete THEN
					AllFBsInitialized := FALSE;
					InfoStations[i].CyclicLogic();
				END_IF
			END_FOR

			IF AllFBsInitialized THEN
				InitializeState := E_XPUInitializeState.eXPUInitializeState_Complete;
			END_IF
		ELSE
			//There will be no station information unless the XPU was initialized
			InitializeState := E_XPUInitializeState.eXPUInitializeState_Complete;
		END_IF

	E_XPUInitializeState.eXPUInitializeState_Complete:
		_State	   := E_XTSState.eXTSState_Disabled;
		Initialize := SUPER^.Initialize();

	E_XPUInitializeState.eXPUInitializeState_Failed:
		IF NOT XPUAlarms[E_XPUAlarms.InitializationError].bRaised THEN
			RaiseAlarm(Alarm := XPUAlarms[E_XPUAlarms.InitializationError]);
		END_IF

		_Busy  := FALSE;
		_Error := TRUE;
END_CASE
END_METHOD

METHOD PRIVATE ClearAllEvents
VAR
	i : UDINT;
END_VAR
FOR i := 1 TO CONSTANTS.XPU_ALARM_COUNT DO
	IF XPUAlarms[i].bRaised THEN
		XPUAlarms[i].Clear(0, 0);
	END_IF
END_FOR
END_METHOD

METHOD CollectRecoveryData
VAR
	i : UDINT;
END_VAR

VAR_INST
	PreviousPersistentRecoveryData : ARRAY[1..TcIoXtsEnvironmentParameterList.MaxXtsInfoServer * TcIoXtsEnvironmentParameterList.MaxXtsInfoStation] OF ST_MoverAssignmentData;
END_VAR
FOR i := 1 TO NumberOfStations DO
	IF InfoStations[i].ipInfoStation <> 0 THEN
		MoverAssignments_NOVRAM[i].StationID := InfoStations[i].ipInfoStation.GetStationId();
		MoverAssignments_NOVRAM[i].MoverIDs	 := InfoStations[i].MoverQueue.MoverIDs;
		MEMCPY(ADR(MoverAssignments_Persistent), ADR(MoverAssignments_NOVRAM), SIZEOF(MoverAssignments_NOVRAM));
	ELSE
		RaiseAlarmWithStrings(XPUAlarms[E_XPUAlarms.NullPointerException], 'CollectRecoveryData()', '');
	END_IF
END_FOR

IF _MoverAssignmentStorageLocation = E_MoverAssignmentRecoverySource.eMoverAssignmentRecoverySource_Persistent THEN
	IF MEMCMP(ADR(PreviousPersistentRecoveryData), ADR(MoverAssignments_Persistent), SIZEOF(MoverAssignments_Persistent)) <> 0 THEN
		IF NOT WritePersistentData.BUSY AND NOT WritePersistentData.ERR THEN
			WritePersistentData.START := TRUE;
		END_IF
	END_IF

	WritePersistentData(PORT := TwinCAT_SystemInfoVarList._AppInfo.AdsPort, MODE := SPDM_2PASS);
	IF NOT WritePersistentData.BUSY THEN
		IF WritePersistentData.ERR THEN
			RaiseAlarmWithStrings(XPUAlarms[E_XPUAlarms.WritePersistentError], TO_STRING(WritePersistentData.ERRID), '');
		END_IF

		WritePersistentData(START := FALSE);
		MEMCPY(ADR(PreviousPersistentRecoveryData), ADR(MoverAssignments_Persistent), SIZEOF(MoverAssignments_Persistent));
	END_IF
END_IF
END_METHOD

METHOD PRIVATE FINAL FindRecoveryCandidates : BOOL
VAR_IN_OUT
	ipCandidates : ARRAY[0..TcIoXtsEnvironmentParameterList.MaxXtsInfoServer * TcIoXtsEnvironmentParameterList.MaxXtsInfoStation] OF I_XTS_InfoStation;
END_VAR

VAR
	StationConfig	   : ST_XTSStationConfig;
	i				   : UDINT;
	NumberOfCandidates : UDINT;
END_VAR
//Check all station configurations and collect all of the queues
FOR i := 1 TO NumberOfStations DO
	IF InfoStations[i].IsAQueue THEN
		NumberOfCandidates				 := NumberOfCandidates + 1;
		ipCandidates[NumberOfCandidates] := InfoStations[i];
	END_IF
END_FOR

IF NumberOfCandidates > 0 THEN
	FindRecoveryCandidates := TRUE;
ELSE
	_Error := TRUE;
END_IF
END_METHOD

METHOD PRIVATE FINAL MoverAssignmentRecovery : BOOL
VAR_INST
	State				 : E_XPUColdStartRecoveryState;
	ipRecoveryCandidates : ARRAY[0..TcIoXtsEnvironmentParameterList.MaxXtsInfoServer * TcIoXtsEnvironmentParameterList.MaxXtsInfoStation] OF I_XTS_InfoStation;
END_VAR
CASE State OF
	E_XPUColdStartRecoveryState.eXPUColdStartRecoveryState_CheckMover1Config:
		IF ipXPU <> 0 THEN
			IF ipXPU.GetMoverIdDetectionMode() = MoverIdDetectionMode.Standard THEN
				IF Parameters_XTS.ENABLE_DEBUG_TRACING THEN
					Trace('Mover 1 detection is not set');
				END_IF

				State := E_XPUColdStartRecoveryState.eXPUColdStartRecoveryState_CheckPersistentDataSource;
			ELSE
				IF Parameters_XTS.ENABLE_DEBUG_TRACING THEN
					Trace('Mover 1 detection is set.  Waiting for drive ready.');
				END_IF

				State := E_XPUColdStartRecoveryState.eXPUColdStartRecoveryState_WaitForDriveReady;
			END_IF
		ELSE
			IF Parameters_XTS.ENABLE_DEBUG_TRACING THEN
				IF Parameters_XTS.ENABLE_DEBUG_TRACING THEN
					Trace('XPU Interface Pointer is NULL');
				END_IF

				RaiseAlarm(Alarm := XPUAlarms[E_XPUAlarms.InitializationError]);
				_Busy  := FALSE;
				_Error := TRUE;
			END_IF
		END_IF

	E_XPUColdStartRecoveryState.eXPUColdStartRecoveryState_WaitForDriveReady:
		IF ipXPU.GetOperationMode() = OperationMode.Normal THEN
			IF Parameters_XTS.ENABLE_DEBUG_TRACING THEN
				Trace('Starting Mover 1 Detection Cycle');
			END_IF

			State := E_XPUColdStartRecoveryState.eXPUColdStartRecoveryState_StartMover1Detection;
		ELSE
			IF Parameters_XTS.ENABLE_DEBUG_TRACING THEN
				Trace('Cannot use Mover 1 in simulation mode');
			END_IF

			RaiseAlarm(Alarm := XPUAlarms[E_XPUAlarms.Mover1DetectionError]);
			_Busy					:= FALSE;
			_Error					:= TRUE;
			State					:= E_XPUColdStartRecoveryState.eXPUColdStartRecoveryState_WaitForDriveReady;
			MoverAssignmentRecovery := TRUE;
		END_IF

	E_XPUColdStartRecoveryState.eXPUColdStartRecoveryState_StartMover1Detection:
		IF ipXPU.TriggerMoverIdDetection() THEN
			IF Parameters_XTS.ENABLE_DEBUG_TRACING THEN
				Trace('Mover 1 Detection Active');
			END_IF

			State := E_XPUColdStartRecoveryState.eXPUColdStartRecoveryState_WaitForMover1DetectionComplete;
		END_IF

	E_XPUColdStartRecoveryState.eXPUColdStartRecoveryState_WaitForMover1DetectionComplete:
		IF ipXPU.GetHasMoverIdDetectionError() THEN
			IF Parameters_XTS.ENABLE_DEBUG_TRACING THEN
				Trace('Mover 1 Detection Error');
			END_IF

			RaiseAlarm(Alarm := XPUAlarms[E_XPUAlarms.Mover1DetectionError]);
			_Busy					:= FALSE;
			_Error					:= TRUE;
			State					:= E_XPUColdStartRecoveryState.eXPUColdStartRecoveryState_WaitForDriveReady;
			MoverAssignmentRecovery := TRUE;
		ELSIF ipXPU.GetIsMoverIdDetectionValid() THEN
			State := E_XPUColdStartRecoveryState.eXPUColdStartRecoveryState_CheckPersistentDataSource;
		END_IF

	E_XPUColdStartRecoveryState.eXPUColdStartRecoveryState_CheckPersistentDataSource:
		CASE _MoverAssignmentStorageLocation OF
			E_MoverAssignmentRecoverySource.eMoverAssignmentRecoverySource_NoBackup:
				IF Parameters_XTS.ENABLE_DEBUG_TRACING THEN
					Trace('No mover assignment backup data');
				END_IF

				State := E_XPUColdStartRecoveryState.eXPUColdStartRecoveryState_LookForRecoveryCandidates;

			E_MoverAssignmentRecoverySource.eMoverAssignmentRecoverySource_Persistent:
				IF Parameters_XTS.ENABLE_DEBUG_TRACING THEN
					Trace('Using persistent data for recovery');
				END_IF

				IF TwinCAT_SystemInfoVarList._AppInfo.BootDataLoaded THEN
					CASE TwinCAT_SystemInfoVarList._AppInfo.PersistentStatus OF
						EPlcPersistentStatus.PS_None, EPlcPersistentStatus.PS_Partial:
							IF Parameters_XTS.ENABLE_DEBUG_TRACING THEN
								Trace('Persistent data did not load properly');
							END_IF

							RaiseAlarm(Alarm := XPUAlarms[E_XPUAlarms.MoverAssignmentRecoveryError]);
							_Busy					:= FALSE;
							_Error					:= TRUE;
							State					:= E_XPUColdStartRecoveryState.eXPUColdStartRecoveryState_LookForRecoveryCandidates;
							MoverAssignmentRecovery := TRUE;

						EPlcPersistentStatus.PS_All:
							State := E_XPUColdStartRecoveryState.eXPUColdStartRecoveryState_RestorePersistentStationMoverAssignments;
					END_CASE
				END_IF

				State := E_XPUColdStartRecoveryState.eXPUColdStartRecoveryState_RestorePersistentStationMoverAssignments;

			e_MoverAssignmentRecoverySource.eMoverAssignmentRecoverySource_NOVRAM:
				IF Parameters_XTS.ENABLE_DEBUG_TRACING THEN
					Trace('Using NOVRAM for recovery data');
				END_IF

				State := E_XPUColdStartRecoveryState.eXPUColdStartRecoveryState_RestoreNOVRAMStationMoverAssignments;
		END_CASE

	E_XPUColdStartRecoveryState.eXPUColdStartRecoveryState_RestorePersistentStationMoverAssignments:
		IF RestoreBackupData(MoverAssignments_Persistent) THEN
			State := E_XPUColdStartRecoveryState.eXPUColdStartRecoveryState_RecoveryComplete;
		ELSIF _Error THEN
			//Restoring persistent backup failed for some reason
			RaiseAlarm(Alarm := XPUAlarms[E_XPUAlarms.MoverAssignmentRecoveryError]);
			_Busy					:= FALSE;
			_Error					:= TRUE;
			State					:= E_XPUColdStartRecoveryState.eXPUColdStartRecoveryState_LookForRecoveryCandidates;
			MoverAssignmentRecovery := TRUE;
		END_IF

	E_XPUColdStartRecoveryState.eXPUColdStartRecoveryState_RestoreNOVRAMStationMoverAssignments:
		IF RestoreBackupData(MoverAssignments_NOVRAM) THEN
			State := E_XPUColdStartRecoveryState.eXPUColdStartRecoveryState_RecoveryComplete;
		ELSIF _Error THEN
			//Restoring NOVRAM backup failed for some reason
			RaiseAlarm(Alarm := XPUAlarms[E_XPUAlarms.MoverAssignmentRecoveryError]);
			_Busy					:= FALSE;
			_Error					:= TRUE;
			State					:= E_XPUColdStartRecoveryState.eXPUColdStartRecoveryState_LookForRecoveryCandidates;
			MoverAssignmentRecovery := TRUE;
		END_IF

	E_XPUColdStartRecoveryState.eXPUColdStartRecoveryState_LookForRecoveryCandidates:
		IF FindRecoveryCandidates(ipRecoveryCandidates) THEN
			State := E_XPUColdStartRecoveryState.eXPUColdStartRecoveryState_ForceMoversOntoCandidates;
		ELSIF _Error THEN
			RaiseAlarm(Alarm := XPUAlarms[E_XPUAlarms.MoverAssignmentRecoveryError]);
			_Busy					:= FALSE;
			_Error					:= TRUE;
			State					:= E_XPUColdStartRecoveryState.eXPUColdStartRecoveryState_LookForRecoveryCandidates;
			MoverAssignmentRecovery := TRUE;
		END_IF

	E_XPUColdStartRecoveryState.eXPUColdStartRecoveryState_ForceMoversOntoCandidates:
		IF ReassignMovers(ipRecoveryCandidates, ipMovers) THEN
			State := E_XPUColdStartRecoveryState.eXPUColdStartRecoveryState_RecoveryComplete;
		ELSIF _Error THEN
			RaiseAlarm(Alarm := XPUAlarms[E_XPUAlarms.MoverAssignmentRecoveryError]);
			_Busy					:= FALSE;
			_Error					:= TRUE;
			State					:= E_XPUColdStartRecoveryState.eXPUColdStartRecoveryState_LookForRecoveryCandidates;
			MoverAssignmentRecovery := TRUE;
		END_IF

	E_XPUColdStartRecoveryState.eXPUColdStartRecoveryState_RecoveryComplete:
		State					:= E_XPUColdStartRecoveryState.eXPUColdStartRecoveryState_LookForRecoveryCandidates;
		StationRecoveryComplete := TRUE;
		MoverAssignmentRecovery := TRUE;
END_CASE
END_METHOD

METHOD PRIVATE FINAL ReassignMovers : BOOL
VAR_IN_OUT
	ipCandidates : ARRAY[0..TcIoXtsEnvironmentParameterList.MaxXtsInfoServer * TcIoXtsEnvironmentParameterList.MaxXtsInfoStation] OF I_XTS_InfoStation;
END_VAR

VAR_INPUT
	ipMovers : ARRAY[0..TcIoXtsEnvironmentParameterList.MaxXtsMoversPerXpu] OF I_XTS_Mover;
END_VAR

VAR_INST
	SequenceState	   : UDINT;
	NumberOfCandidates : UDINT;
	MoverBuckets	   : ARRAY[1..TcIoXtsEnvironmentParameterList.MaxXtsInfoServer * TcIoXtsEnvironmentParameterList.MaxXtsInfoStation, 0..TcIoXtsEnvironmentParameterList.MaxXtsMoversPerXpu] OF
		I_XTS_Mover;
	MoversHandled : UDINT;
END_VAR

VAR
	i, j								 : UDINT;
	temp								 : I_XTS_InfoStation;
	StationPosition_i, StationPosition_j : LREAL;
	MoversInBucket						 : UDINT;
END_VAR
CASE SequenceState OF
	0:
		NumberOfCandidates := 0;
		MEMSET(ADR(MoverBuckets), 0, SIZEOF(MoverBuckets));

		//Find the number of candidates
		FOR i := 1 TO TcIoXtsEnvironmentParameterList.MaxXtsInfoServer * TcIoXtsEnvironmentParameterList.MaxXtsInfoStation DO
			IF ipCandidates[i] <> 0 THEN
				NumberOfCandidates := NumberOfCandidates + 1;
			ELSE
				EXIT;
			END_IF
		END_FOR

		IF NumberOfCandidates > 0 THEN
			SequenceState := SequenceState + 10;
		ELSE
			;
			//TODO: Flag error here
		END_IF

	10:
		//Sort Stations
		FOR i := 1 TO NumberOfCandidates DO
			StationPosition_i := ipCandidates[i].GetStopPositionOnTrack(ipCandidates[i].ApplicationStation.TrackOID, ipCandidates[i].StopPositions[1]);
			FOR j := i + 1 TO NumberOfCandidates DO
				StationPosition_j := ipCandidates[j].GetStopPositionOnTrack(ipCandidates[j].ApplicationStation.TrackOID, ipCandidates[j].StopPositions[1]);
				IF (StationPosition_i > StationPosition_j) THEN
					temp			:= ipCandidates[i];
					ipCandidates[i] := ipCandidates[j];
					ipCandidates[j] := temp;
				END_IF
			END_FOR
		END_FOR

		SequenceState := SequenceState + 10;

	20:
		MoversHandled := 0;

		//Put movers in buckets
		FOR i := 1 TO NumberOfCandidates DO
			MoversInBucket	  := 0;
			StationPosition_i := ipCandidates[i].GetStopPositionOnTrack(ipCandidates[i].ApplicationStation.TrackOID, ipCandidates[i].StopPositions[1]);
			FOR j := 1 TO NumberOfMovers DO
				IF ipMovers[j] <> 0 THEN
					IF ipMovers[j].SetPositionModulo <= StationPosition_i THEN
						MoversInBucket					:= MoversInBucket + 1;
						MoverBuckets[i, MoversInBucket] := ipMovers[j];
						ipMovers[j]						:= 0;
						MoversHandled					:= MoversHandled + 1;
					END_IF
				END_IF
			END_FOR
		END_FOR

		//We are going to put any remaining unassigned movers into the first station's bucket so need the count
		MoversInBucket := 0;
		FOR i := 1 TO NumberOfMovers DO
			IF MoverBuckets[1, i] <> 0 THEN
				MoversInBucket := MoversInBucket + 1;
			ELSE
				EXIT;
			END_IF
		END_FOR

		//Put any remaining unassigned movers into the first station's bucket
		FOR i := 1 TO NumberOfMovers DO
			IF ipMovers[i] <> 0 THEN
				MoversInBucket					:= MoversInBucket + 1;
				MoverBuckets[1, MoversInBucket] := ipMovers[i];
				ipMovers[i]						:= 0;
			END_IF
		END_FOR

		SequenceState := SequenceState + 10;

	30:
		IF SortMoverBuckets(ipCandidates, MoverBuckets, NumberOfCandidates) THEN
			SequenceState := SequenceState + 10;
		END_IF

	40:
		FOR i := 1 TO NumberOfCandidates DO
			FOR j := 1 TO NumberOfMovers DO
				IF MoverBuckets[i, j] <> 0 THEN
					ipCandidates[i].MoverQueue.Enqueue(MoverBuckets[i, j]);
				ELSE
					EXIT;
				END_IF
			END_FOR
		END_FOR

		SequenceState  := 0;
		ReassignMovers := TRUE;
END_CASE
END_METHOD

METHOD PRIVATE RestoreBackupData : BOOL;
VAR_INPUT
	Backup : ARRAY[1..TcIoXtsEnvironmentParameterList.MaxXtsInfoServer * TcIoXtsEnvironmentParameterList.MaxXtsInfoStation] OF ST_MoverAssignmentData;
END_VAR

VAR
	i, j, k, l		: UDINT;
	MoversRestored	: UDINT;
	DoneWithStation : BOOL;
END_VAR
FOR i := 1 TO TcIoXtsEnvironmentParameterList.MaxXtsInfoServer * TcIoXtsEnvironmentParameterList.MaxXtsInfoStation DO
	DoneWithStation := FALSE;

	//Iterate through all possible backup data
	IF Backup[i].StationID = 0 THEN
		//Nothing was backed up here
		EXIT;
	END_IF

	FOR j := 1 TO TcIoXtsEnvironmentParameterList.MaxXtsInfoServer * TcIoXtsEnvironmentParameterList.MaxXtsInfoStation DO
		//Match infostation ID with backup location ID
		IF InfoStations[j].StationID = 0 OR DoneWithStation THEN
			//There is no infostation in this location
			EXIT;
		ELSIF InfoStations[j].StationID = Backup[i].StationID THEN
			//InfoStation[j] matches this backup location OID
			FOR k := 1 TO TcIoXtsEnvironmentParameterList.MaxXtsMoversPerXpu DO
				IF Backup[i].MoverIDs[k] = 0 THEN
					//MoverIDs should be start at index 1 so if encountering zero there are none left
					DoneWithStation := TRUE;
					EXIT;
				ELSE
					DoneWithStation := TRUE;
					FOR l := 1 TO TcIoXtsEnvironmentParameterList.MaxXtsMoversPerXpu DO
						//Iterate though all possible movers and match mover ID to backup mover ID
						IF Movers[l].MoverID = Backup[i].MoverIDs[k] THEN
							//This mover belongs with this station--enqueue it.
							InfoStations[j].MoverQueue.Enqueue(Movers[l]);
							MoversRestored := MoversRestored + 1;
							EXIT;
						END_IF
					END_FOR
				END_IF
			END_FOR
		END_IF
	END_FOR
END_FOR

IF MoversRestored = NumberOfMovers THEN
	RestoreBackupData := TRUE;
ELSE
	_Error := TRUE;
END_IF
END_METHOD

METHOD PRIVATE FINAL SetError : BOOL
VAR_INPUT
	ErrorID : UDINT;
END_VAR

//VAR

//    i : UDINT;

//END_VAR
_Busy		  := FALSE;
_Error		  := TRUE;
_ErrorID	  := ErrorID;
SequenceState := 0;
_State		  := E_XTSState.eXTSState_Error;
END_METHOD

METHOD FINAL SetStationNeighbors
VAR
	i : UDINT;
END_VAR
FOR i := 1 TO NumberOfStations DO
	StationNeigbors[i].Station := InfoStations[i];
	IF i = 1 THEN
		//First station's previous neighbor is the last station
		StationNeigbors[i].UpstreamStation := InfoStations[NumberOfStations];
		IF NumberOfStations > 1 THEN
			StationNeigbors[i].DownstreamStation := InfoStations[i + 1];
		ELSE
			//Weird case where there is only one station
			StationNeigbors[i].DownstreamStation := InfoStations[1];
		END_IF
	ELSE
		StationNeigbors[i].UpstreamStation := InfoStations[i - 1];
		IF i = NumberOfStations THEN
			StationNeigbors[i].DownstreamStation := InfoStations[1];
		ELSE
			StationNeigbors[i].DownstreamStation := InfoStations[i + 1];
		END_IF
	END_IF
END_FOR
END_METHOD

METHOD SortMoverBuckets : BOOL
VAR_IN_OUT
	ipCandidates : ARRAY[0..TcIoXtsEnvironmentParameterList.MaxXtsInfoServer * TcIoXtsEnvironmentParameterList.MaxXtsInfoStation] OF I_XTS_InfoStation;
	MoverBuckets : ARRAY[1..TcIoXtsEnvironmentParameterList.MaxXtsInfoServer * TcIoXtsEnvironmentParameterList.MaxXtsInfoStation, 0..TcIoXtsEnvironmentParameterList.MaxXtsMoversPerXpu] OF
		I_XTS_Mover;
END_VAR

VAR_INPUT
	NumberOfCandidates : UDINT;
END_VAR

VAR
	i, j			 : UDINT;
	CurrentCandidate : UDINT;
	StationPosition	 : LREAL;
	UnsortedBucket	 : ARRAY[0..TcIoXtsEnvironmentParameterList.MaxXtsMoversPerXpu] OF I_XTS_Mover;
	SortedBucket	 : ARRAY[0..TcIoXtsEnvironmentParameterList.MaxXtsMoversPerXpu] OF I_XTS_Mover;
	MoversInBucket	 : UDINT;
	temp			 : I_XTS_Mover;
END_VAR
FOR CurrentCandidate := 1 TO NumberOfCandidates DO
	StationPosition := ipCandidates[CurrentCandidate].GetStopPositionOnTrack(ipCandidates[CurrentCandidate].ApplicationStation.TrackOID, ipCandidates[CurrentCandidate].StopPositions[1]);
	MEMCPY(ADR(UnsortedBucket), ADR(MoverBuckets[CurrentCandidate, 0]), SIZEOF(UnsortedBucket));
	MEMSET(ADR(MoverBuckets[CurrentCandidate, 0]), 0, SIZEOF(UnsortedBucket));
	MoversInBucket := 0;

	//Count the number of movers in this bucket
	FOR i := 1 TO TcIoXtsEnvironmentParameterList.MaxXtsMoversPerXpu DO
		IF UnsortedBucket[i] <> 0 THEN
			MoversInBucket := MoversInBucket + 1;
		ELSE
			EXIT;
		END_IF
	END_FOR

	IF MoversInBucket > 1 THEN
		//Sort the bucket in descending order
		FOR i := 1 TO MoversInBucket DO
			FOR j := i + 1 TO MoversInBucket DO
				IF (UnsortedBucket[i].SetPositionModulo < UnsortedBucket[j].SetPositionModulo) THEN
					temp			  := UnsortedBucket[i];
					UnsortedBucket[i] := UnsortedBucket[j];
					UnsortedBucket[j] := temp;
				END_IF
			END_FOR
		END_FOR

		FOR i := 1 TO (MoversInBucket - 1) DO
			IF UnsortedBucket[1].SetPositionModulo > StationPosition THEN
				temp := UnsortedBucket[1];
				MEMSET(ADR(UnsortedBucket[1]), 0, SIZEOF(UnsortedBucket[1]));
				MEMCPY(ADR(UnsortedBucket[1]), ADR(UnsortedBucket[2]), SIZEOF(UnsortedBucket[1]) * (MoversInBucket - 1));
				MEMSET(ADR(UnsortedBucket[MoversInBucket]), 0, SIZEOF(UnsortedBucket[i]));
				MEMCPY(ADR(UnsortedBucket[MoversInBucket]), ADR(temp), SIZEOF(temp));
			END_IF
		END_FOR
	END_IF

	MEMCPY(ADR(MoverBuckets[CurrentCandidate, 0]), ADR(UnsortedBucket), SIZEOF(UnsortedBucket));
END_FOR

SortMoverBuckets := TRUE;
END_METHOD

METHOD FINAL Trace
VAR_INPUT
	Message : T_MaxString;
END_VAR

VAR
	Document	  : SJsonValue;
	XTSJsonObject : SJsonValue;
	StateString	  : T_MaxString;
	JsonAttribute : T_MaxString;
END_VAR
{analysis -62}
StateString := TO_STRING(_State);
Document	:= JsonParser.NewDocument();
JsonParser.AddObjectMember(Document, 'XTS');
XTSJsonObject := JsonParser.FindMember(Document, 'XTS');
JsonParser.AddStringMember(XTSJsonObject, 'XTSId', _Name);
JsonParser.AddUintMember(XTSJsonObject, 'Movers', NumberOfMovers);
JsonParser.AddUintMember(XTSJsonObject, 'Stations', NumberOfStations);
JsonParser.AddStringMember(XTSJsonObject, 'State', StateString);
TraceWithJson(Message, JsonParser.GetJson(Document));
END_METHOD

METHOD PUBLIC ClearMoverAssignments : BOOL
VAR
	i : UDINT;
END_VAR
IF _State = E_XTSState.eXTSState_Disabled OR _State = E_XTSState.eXTSState_Error THEN
	FOR i := 1 TO NumberOfStations DO
		InfoStations[i].ReleaseAllMovers();
	END_FOR

	MEMSET(ADR(MoverAssignments_Persistent), 0, SIZEOF(MoverAssignments_Persistent));
	MEMSET(ADR(MoverAssignments_NOVRAM), 0, SIZEOF(MoverAssignments_NOVRAM));
	InitializeState			:= E_XPUInitializeState.eXPUInitializeState_AttemptMoverRecovery;
	StationRecoveryComplete := FALSE;
	SequenceState			:= 0;
	ClearMoverAssignments	:= TRUE;
END_IF
END_METHOD

METHOD PUBLIC Disable : BOOL
VAR
	i : UDINT;
END_VAR
CASE SequenceState OF
	0:
		IF _State = E_XTSState.eXTSState_Enabled THEN
			_State := E_XTSState.eXTSState_Disabling;
			Trace('XPU Disable Requested');
			_Busy := TRUE;
			MoverTracker.Clear();
			SequenceState := SequenceState + 10;
		END_IF

	10:
		//Stop the CA group
		MCGroupStop(AxesGroup := CAGroup, Execute := TRUE);
		IF MCGroupReadStatus.GroupErrorStop THEN
			MCGroupStop(AxesGroup := CAGroup, Execute := FALSE);
			SetError(MCGroupReadError.GroupErrorId);
		ELSIF MCGroupStop.Error THEN
			MCGroupStop(AxesGroup := CAGroup, Execute := FALSE);
			SetError(MCGroupStop.ErrorID);
		ELSIF MCGroupStop.Done OR MCGroupReadStatus.AllAxesStanding THEN
			MCGroupStop(AxesGroup := CAGroup, Execute := FALSE);
			SequenceState := SequenceState + 10;
		END_IF

	20:
		//Disable the CA group
		MCGroupDisable(AxesGroup := CAGroup, Execute := TRUE);
		IF MCGroupReadStatus.GroupErrorStop THEN
			MCGroupDisable(AxesGroup := CAGroup, Execute := FALSE);
			SetError(MCGroupReadError.GroupErrorId);
		ELSIF MCGroupDisable.Error THEN
			MCGroupDisable(AxesGroup := CAGroup, Execute := FALSE);
			SetError(MCGroupDisable.ErrorID);
		ELSIF MCGroupDisable.Done OR MCGroupReadStatus.GroupDisabled THEN
			MCGroupDisable(AxesGroup := CAGroup, Execute := FALSE);
			SequenceState := SequenceState + 10;
		END_IF

	30:
		//Dissolve the CA group
		MCUngroupAllAxes(AxesGroup := CAGroup, Execute := TRUE);
		IF MCGroupReadStatus.GroupErrorStop THEN
			MCUngroupAllAxes(AxesGroup := CAGroup, Execute := FALSE);
			SetError(MCGroupReadError.GroupErrorId);
		ELSIF MCUngroupAllAxes.Error THEN
			MCUngroupAllAxes(AxesGroup := CAGroup, Execute := FALSE);
			SetError(MCUngroupAllAxes.ErrorID);
		ELSIF MCUngroupAllAxes.Done THEN
			MCUngroupAllAxes(AxesGroup := CAGroup, Execute := FALSE);
			SequenceState := SequenceState + 10;
		END_IF

	40:
		//Disable all mover axes
		FOR i := 1 TO NumberOfMovers DO
			IF NOT MoverTracker.Check(i) AND_THEN ipMovers[i].Disable() THEN
				MoverTracker.Set(i);
			END_IF
		END_FOR

		IF MoverTracker.NumberCompleted = NumberOfMovers THEN
			MoverTracker.Clear();
			SequenceState := SequenceState + 10;
		END_IF

	50:
		//Check all mover axes are disabled
		FOR i := 1 TO NumberOfMovers DO
			IF NOT ipMovers[i].Busy THEN
				IF ipMovers[i].Error THEN
					SetError(ipMovers[i].ErrorID);
				ELSE
					MoverTracker.Set(i);
				END_IF
			END_IF
		END_FOR

		IF MoverTracker.NumberCompleted = NumberOfMovers THEN
			MoverTracker.Clear();
			Trace('XPU Disable Completed');
			SequenceState := 1000;
		END_IF

	1000:
		_State		  := E_XTSState.eXTSState_Disabled;
		SequenceState := 0;
		Disable		  := TRUE;
END_CASE
END_METHOD

METHOD PUBLIC Enable : BOOL
VAR
	i : UDINT;
END_VAR
CASE SequenceState OF
	0:
		IF _State = E_XTSState.eXTSState_Disabled THEN
			_State := E_XTSState.eXTSState_Enabling;
			Trace('XPU Enable Requested');
			_Busy := TRUE;
			MoverTracker.Clear();
			SequenceState := SequenceState + 10;
		END_IF

	10:
		//Enable all movers
		FOR i := 1 TO NumberOfMovers DO
			IF NOT MoverTracker.Check(i) AND_THEN ipMovers[i].Enable() THEN
				MoverTracker.Set(i);
			END_IF
		END_FOR

		IF MoverTracker.NumberCompleted = NumberOfMovers THEN
			MoverTracker.Clear();
			SequenceState := SequenceState + 10;
		END_IF

	20:
		//Check all movers were enabled
		FOR i := 1 TO NumberOfMovers DO
			IF NOT ipMovers[i].Busy THEN
				IF ipMovers[i].Error THEN
					SetError(ipMovers[i].ErrorID);
				ELSIF ipMovers[i].Enabled THEN
					MoverTracker.Set(i);
				END_IF
			END_IF
		END_FOR

		IF MoverTracker.NumberCompleted = NumberOfMovers THEN
			MoverTracker.Clear();
			SequenceState := SequenceState + 10;
		END_IF

	30:
		//Add all movers to CA group
		FOR i := 1 TO NumberOfMovers DO
			IF NOT MoverTracker.Check(i) AND_THEN ipMovers[i].JoinGroup() THEN
				MoverTracker.Set(i);
			END_IF
		END_FOR

		IF MoverTracker.NumberCompleted = NumberOfMovers THEN
			MoverTracker.Clear();
			SequenceState := SequenceState + 10;
		END_IF

	40:
		//Check all movers were added to CA group
		FOR i := 1 TO NumberOfMovers DO
			IF NOT ipMovers[i].Busy THEN
				IF ipMovers[i].Error THEN
					SetError(ipMovers[i].ErrorID);
				ELSE
					MoverTracker.Set(i);
				END_IF
			END_IF
		END_FOR

		IF MoverTracker.NumberCompleted = NumberOfMovers THEN
			MoverTracker.Clear();
			SequenceState := SequenceState + 10;
		END_IF

	50:
		//Enable CA group
		MCGroupEnable(AxesGroup := CAGroup, Execute := TRUE);
		IF NOT MCGroupEnable.Busy THEN
			IF MCGroupReadStatus.GroupErrorStop THEN
				SetError(MCGroupReadError.GroupErrorId);
			ELSIF MCGroupEnable.Error THEN
				SetError(MCGroupEnable.ErrorID);
			ELSIF MCGroupEnable.Done THEN
				Trace('XPU Enable Completed');
				SequenceState := 1000;
			END_IF

			MCGroupEnable(AxesGroup := CAGroup, Execute := FALSE);
		END_IF

	1000:
		_State		  := E_XTSState.eXTSState_Enabled;
		SequenceState := 0;
		Enable		  := TRUE;
END_CASE
END_METHOD

METHOD FB_init : BOOL
VAR_INPUT
	bInitRetains : BOOL; // if TRUE, the retain variables are initialized (warm start / cold start)
	bInCopyCode	 : BOOL; // if TRUE, the instance afterwards gets moved into the copy code (online change)
END_VAR

VAR
	i : UDINT;
END_VAR
FOR i := 1 TO TcIoXtsEnvironmentParameterList.MaxXtsPartsPerXpu DO
	Parts[i].ipXPU := THIS^;
END_FOR

FOR i := 1 TO TcIoXtsEnvironmentParameterList.MaxXtsMoversPerXpu DO
	Movers[i].Group REF= CAGroup;
	ipMovers[i]		:= Movers[i];
END_FOR

StationTracker.StationsToTrack REF= NumberOfStations;
END_METHOD

PROPERTY MoverAssignmentStorageLocation : E_MoverAssignmentRecoverySource
GET
MoverAssignmentStorageLocation := _MoverAssignmentStorageLocation;
END_GET
SET
_MoverAssignmentStorageLocation := MoverAssignmentStorageLocation;
END_SET
END_PROPERTY

PROPERTY PartCoEData : ARRAY[1..TcIoXtsEnvironmentParameterList.MaxXtsPartsPerXpu] OF ARRAY[1..TcIoXtsEnvironmentParameterList.MaxModulesPerPart] OF ST_AT2xxxAllCoEData
GET
PartCoEData := _PartCoEData;
END_GET
END_PROPERTY

METHOD PUBLIC Reset : BOOL
VAR
	i			   : UDINT;
	AllOpsComplete : BOOL;
END_VAR
//IF _State = E_XTSState.eXTSState_Error OR _State = E_XTSState.eXTSState_Reset THEN
CASE SequenceState OF
	0:
		_State := E_XTSState.eXTSState_Reset;
		Trace('XPU Reset Requested');
		_Busy := TRUE;
		MoverTracker.Clear();
		IF ipXPU.GetIsPartBasedHandlingActivated() THEN
			SequenceState := 1;
		ELSE
			SequenceState := 10;
		END_IF

	1:
		AllOpsComplete := TRUE;
		FOR i := 1 TO NumberOfParts DO
			IF Parts[i].Error THEN
				AllOpsComplete := Parts[i].Reset();
			END_IF
		END_FOR

		IF AllOpsComplete THEN
			SequenceState := 2;
		END_IF

	2:
		AllOpsComplete := TRUE;
		FOR i := 1 TO NumberOfParts DO
			IF Parts[i].Error THEN
				AllOpsComplete := FALSE;
			END_IF
		END_FOR

		IF AllOpsComplete THEN
			SequenceState := 10;
		ELSE
			SequenceState := 1000;
		END_IF

	10:
		FOR i := 1 TO NumberOfMovers DO
			IF NOT MoverTracker.Check(i) AND_THEN ipMovers[i].Disable() THEN
				ipMovers[i].LimitBipolarCurrent := FALSE;
				MoverTracker.Set(i);
			END_IF
		END_FOR

		IF MoverTracker.NumberCompleted = NumberOfMovers THEN
			MoverTracker.Clear();
			SequenceState := SequenceState + 10;
		END_IF

	20:
		FOR i := 1 TO NumberOfMovers DO
			IF NOT ipMovers[i].Busy THEN
				MoverTracker.Set(i);
			END_IF
		END_FOR

		IF MoverTracker.NumberCompleted = NumberOfMovers THEN
			MoverTracker.Clear();
			SequenceState := SequenceState + 10;
		END_IF

	30:
		// Reset collision avoidance group
		MCGroupReset(AxesGroup := CAGroup, Execute := TRUE);
		IF NOT MCGroupReset.Busy THEN
			IF MCGroupReset.Error THEN
				SetError(MCGroupEnable.ErrorID);
			ELSIF MCGroupReset.Done THEN
				SequenceState := SequenceState + 10;
			END_IF

			MCGroupReset(AxesGroup := CAGroup, Execute := FALSE);
		END_IF

	40:
		FOR i := 1 TO NumberOfMovers DO
			IF NOT MoverTracker.Check(i) AND_THEN (NOT ipMovers[i].Error) OR_ELSE (ipMovers[i].Reset()) THEN
				MoverTracker.Set(i);
			END_IF
		END_FOR

		IF MoverTracker.NumberCompleted = NumberOfMovers THEN
			MoverTracker.Clear();
			SequenceState := SequenceState + 10;
		END_IF

	50:
		FOR i := 1 TO NumberOfMovers DO
			IF NOT ipMovers[i].Busy THEN
				IF ipMovers[i].Error THEN
					SetError(ipMovers[i].ErrorID);
				ELSE
					MoverTracker.Set(i);
				END_IF
			END_IF
		END_FOR

		IF MoverTracker.NumberCompleted = NumberOfMovers THEN
			MoverTracker.Clear();
			Trace('XPU Reset Completed');
			SequenceState := 60;
		END_IF

	60:
		IF StationRecoveryComplete THEN
			SequenceState := 1000;
		ELSE
			SequenceState := SequenceState + 10;
		END_IF

	70:
		IF MoverAssignmentRecovery() THEN
			IF StationRecoveryComplete THEN
				SequenceState := 1000;
			ELSE
				SequenceState := 0;
				SetError(0);
				RaiseAlarm(Alarm := XPUAlarms[E_XPUAlarms.MoverAssignmentRecoveryError]);
				Reset := TRUE;
			END_IF
		END_IF

	1000:
		IF MCGroupReadStatus.GroupDisabled THEN
			_State := E_XTSState.eXTSState_Disabled;
		ELSE
			_State := E_XTSState.eXTSState_Disabled;
		END_IF

		ClearAllEvents();
		SequenceState := 0;
		_Error		  := FALSE;
		_ErrorID	  := 0;
		Reset		  := TRUE;
END_CASE
END_METHOD

PROPERTY State : E_XTSState
GET
State := _State;
END_GET
END_PROPERTY

PROPERTY Stations : ARRAY[0..TcIoXtsEnvironmentParameterList.MaxXtsInfoServer * TcIoXtsEnvironmentParameterList.MaxXtsInfoStation] OF I_XTS_ApplicationStation;
GET
Stations := ipStations;
END_GET
SET
ipStations := Stations;
END_SET
END_PROPERTY

END_FUNCTION_BLOCK
